// TwinCAT 3 PLC project Untitled1
// ProgramVersion: 3.1.4024.0
// libraries:
//   Tc2_Standard, * (Beckhoff Automation GmbH)
//   Tc2_System, * (Beckhoff Automation GmbH)
//   Tc3_Module, * (Beckhoff Automation GmbH)
// project tree:
//   GVLs/ GVL_IO.TcGVL
//   / PlcTask.TcTTO
//   POUs/ MAIN.TcPOU
// real-time tasks:
//   TASK PlcTask: cycle T#10ms, priority 20, ADS port 350
// I/O:
//   DEVICE Device 2 (EtherCAT), AmsNetId 169.254.197.213.3.1
//     Term 1 (EK1100) [EK1100 EtherCAT Coupler (2A E-Bus)]
//       Term 2 (EL1008) [EL1008 8Ch. Dig. Input 24V, 3ms]
//       Term 3 (EL3064) [EL3064 4Ch. Ana. Input 0-10V]
//       Term 4 (EL4034) [EL4034 4Ch. Ana. Output +/-10V, 12bit]
//       Term 5 (EL9011) [EL9011 End Terminal]
// variable links:
//   Untitled1/Untitled1 Instance <-> Device 2 (EtherCAT)/Term 1 (EK1100)/Term 2 (EL1008)
//     PlcTask Inputs/GVL_IO.bDoorInerlock <-> Channel 5/GVL_IO.bDoorInerlock
//     PlcTask Inputs/GVL_IO.bLeftPinLockSens <-> Channel 3/GVL_IO.bLeftPinLockSens
//     PlcTask Inputs/GVL_IO.bLeftPistonSens <-> Channel 2/GVL_IO.bLeftPistonSens
//     PlcTask Inputs/GVL_IO.bRightPinLockSens <-> Channel 4/GVL_IO.bRightPinLockSens
//     PlcTask Inputs/GVL_IO.nRightPistonSens <-> Channel 1/GVL_IO.nRightPistonSens
//   Untitled1/Untitled1 Instance <-> Device 2 (EtherCAT)/Term 1 (EK1100)/Term 3 (EL3064)
//     PlcTask Inputs/GVL_IO.rCurrentHW <-> AI Standard Channel 1/GVL_IO.rCurrentHW
//   Untitled1/Untitled1 Instance <-> Device 2 (EtherCAT)/Term 1 (EK1100)/Term 4 (EL4034)
//     PlcTask Outputs/GVL_IO.iMotorPowerHW <-> AO Outputs Channel 2/GVL_IO.iMotorPowerHW
//     PlcTask Outputs/GVL_IO.iSetPistonsPressureHW <-> AO Outputs Channel 1/GVL_IO.iSetPistonsPressureHW

CONFIGURATION Untitled1
    RESOURCE PLC ON TwinCAT3
        TASK PlcTask(INTERVAL := T#10ms, PRIORITY := 20);
        PROGRAM MAIN WITH PlcTask : MAIN;
    END_RESOURCE
END_CONFIGURATION

// ---- GVLs/GVL_IO.TcGVL

VAR_GLOBAL
	rCurrentHW				AT%I*	:	INT;
	iPistonsPressureHW		AT%I* 	:	INT;
	bRightPinLockSens		AT%I*	:	BOOL;
	bLeftPinLockSens		AT%I*	:	BOOL;
	bLeftPistonSens			AT%I*	: 	BOOL;
	nRightPistonSens		AT%I*	:	BOOL;
	bDoorInerlock			AT%I*	:	BOOL;
	
	iSetPistonsPressureHW	AT%Q* 	:	INT;
	iMotorPowerHW			AT%Q*	:	INT;
	iLeftPinForce			AT%I* 	:	INT;
	iRightPinForce			AT%I* 	:	INT;
	
END_VAR

// ---- POUs/MAIN.TcPOU
PROGRAM MAIN
VAR
	ProcessTime			:	TON;
	RunTimer			:	TON;
	StopTimer			:	TON;
	HoldTimer			:	TON;
	
	iHighPower			: 	INT;
	iHoldPower			: 	INT;
	TestState			:	INT;
	CSVstate			:	INT;
	iMotorPower			:	INT;
	iTestCounter		:	INT;
	iCycleToRun			:	UDINT;
	iPistonsPressure	:	INT;
	
	bStartTest			:	BOOL;
	bStopTest			:	BOOL;
	bTimeoutError		: 	BOOL;
	bProcessEndAtPins	: 	BOOL;
	bProcessEndAtTimeout: 	BOOL;
	bAutomatedOperation	:	BOOL;
	bWriteDataEnd		: 	BOOL;
	bReadyToRun			: 	BOOL;
	
	rMotorCurrenr		:	REAL;
	rRecordMotorCurrenr	:	REAL; //csv
	rTimeToStop			: 	REAL;
	rHMI_MotorCurrent	: 	REAL;// By mA
	rRightPinForce		:	REAL;
	rLeftPinForce		:	REAL;
	iPistonsForceHMI	:	INT;
	
	
	
	arrCurrentMessure	:	ARRAY[1..100] OF REAL;
	arrLeftPinMessure	:	ARRAY[1..100] OF REAL;
	arrRightPinMessure	:	ARRAY[1..100] OF REAL;
	i					:	INT;

	sDataToWrite		:	STRING[500];
	fbFileOpen      	: 	FB_FileOpen;
	fbFileWrite      	:	FB_FileWrite;
	fbFileClose       	: 	FB_FileClose;
	bKeepRuningTests: BOOL;
END_VAR

IF bDoorInerlock THEN
	RunTest();
	SaveData();
END_IF

iSetPistonsPressureHW:=REAL_TO_INT(INT_TO_REAL(iPistonsForceHMI)*32.59);
rMotorCurrenr:=(INT_TO_REAL(rCurrentHW)/32767.0)*15.0;
rHMI_MotorCurrent:=rMotorCurrenr*1000;
iMotorPowerHW:=real_to_int((INT_TO_REAL(iMotorPower)/100)*16383);

ACTION RunTest:
ProcessTime(IN:= , PT:=T#2500MS , Q=> , ET=> );
RunTimer(IN:= , PT:=T#450MS , Q=> , ET=> );
StopTimer(IN:= , PT:=T#50MS , Q=> , ET=> );
HoldTimer(IN:= , PT:=T#2S , Q=> , ET=> );
IF TestState=0 AND CSVstate=0 THEN
	bReadyToRun:=TRUE;
ELSE 
	bReadyToRun:=FALSE;
END_IF
IF iTestCounter<=iCycleToRun THEN
	bKeepRuningTests:=TRUE;
ELSE
	bKeepRuningTests:=FALSE;	
END_IF



CASE TestState OF
	0://standby
		ProcessTime.IN:=FALSE;
		IF bStartTest AND NOT bStopTest AND bLeftPistonSens AND nRightPistonSens THEN
			IF NOT bAutomatedOperation THEN
				bStartTest:=FALSE;
			END_IF
			iTestCounter:=iTestCounter+1;
			ProcessTime.IN:=TRUE;
			bProcessEndAtPins:=FALSE;
			bProcessEndAtTimeout:=FALSE;
			//bReadyToRun:=FALSE;
			i:=1;
			TestState:=10;
		END_IF
	
	10:// start movment and reach pins lock sensors
		arrCurrentMessure[i]:=rMotorCurrenr;
		arrLeftPinMessure[i]:=iLeftPinForce;
		arrRightPinMessure[i]:=iRightPinForce;
		i:=i+1;
		IF i>100 THEN
			i:=1;
		END_IF
		RunTimer.IN:=TRUE;
		iMotorPower:=iHighPower;
		
		IF bLeftPinLockSens AND bRightPinLockSens THEN
			bProcessEndAtPins:=TRUE;
			RunTimer.IN:=FALSE;
			iMotorPower:=iHoldPower;	
			//StopTimer.IN:=TRUE;			
			TestState:=20;
		ELSIF RunTimer.Q THEN
			bProcessEndAtTimeout:=TRUE;
			RunTimer.IN:=FALSE;
			iMotorPower:=0;				
			TestState:=40;
		END_IF	
		
	20: //hols pins in open position for 2 sec
		HoldTimer.IN:=TRUE;
		IF HoldTimer.Q THEN
			iMotorPower:=0;
			TestState:=30;
			FOR i:=i TO i-5 DO
				rRecordMotorCurrenr:=(rRecordMotorCurrenr+arrCurrentMessure[i])/5;
				rRightPinForce:=(rRightPinForce+arrLeftPinMessure[i])/5;	
				rLeftPinForce:=(rLeftPinForce+arrRightPinMessure[i])/5;	
			END_FOR			
		END_IF

		
	
	30:// end movment, release motor until pins in close position
		IF bLeftPistonSens AND nRightPistonSens THEN
			rTimeToStop:=TIME_TO_REAL(StopTimer.ET);
			TestState:=40;
		END_IF

	40:// write data to csv
		IF bWriteDataEnd THEN
			TestState:=0;
		END_IF
END_CASE

IF ProcessTime.Q THEN
	bTimeoutError:=TRUE;
ELSE
	bTimeoutError:=FALSE;	
END_IF
END_ACTION

ACTION SaveData:
sDataToWrite:=concat(REAL_TO_STRING(rRightPinForce),concat(',',concat(REAL_TO_STRING(rLeftPinForce),concat(',',concat(REAL_TO_STRING(rRecordMotorCurrenr),concat(',',concat(REAL_TO_STRING(rTimeToStop),concat(',',concat(BOOL_TO_STRING(bProcessEndAtPins),concat(',',concat(INT_TO_STRING(iPistonsForceHMI),'$N')))))))))));
fbFileOpen(
	sNetId:='' , 
	sPathName:='C:\Users\Administrator\Desktop\Logs\Tests.csv ', // add controller path
	nMode:=FOPEN_MODEAPPEND , 
	ePath:= , 
	bExecute:= , 
	tTimeout:=T#3S , 
	bBusy=> , 
	bError=> , 
	nErrId=> , 
	hFile=> );
fbFileWrite(
	sNetId:='' , 
	hFile:=fbFileOpen.hFile , 
	pWriteBuff:=ADR(sDataToWrite) , 
	cbWriteLen:=LEN(sDataToWrite) , 
	bExecute:= , 
	tTimeout:=T#3S , 
	bBusy=> , 
	bError=> , 
	nErrId=> , 
	cbWrite=> );
fbFileClose(
	sNetId:='' , 
	hFile:=fbFileOpen.hFile , 
	bExecute:= , 
	tTimeout:=T#3S , 
	bBusy=> , 
	bError=> , 
	nErrId=> );			

CASE CSVstate OF
	0://standby
	fbFileOpen.bExecute:=FALSE;
	fbFileWrite.bExecute:=FALSE;
	fbFileClose.bExecute:=FALSE;
		IF TestState=40 THEN
			CSVstate:=10;
		END_IF
	10:// open file
		fbFileOpen.bExecute:=TRUE;
		IF fbFileOpen.bBusy AND NOT fbFileOpen.bError THEN
			CSVstate:=15;
		END_IF	
	15:		
		IF NOT fbFileOpen.bError AND NOT fbFileOpen.bBusy THEN
			CSVstate:=20;
		END_IF	
	20:// write data
		fbFileWrite.bExecute:=TRUE;
		IF fbFileWrite.bBusy AND NOT fbFileWrite.bError THEN
			CSVstate:=25;
		END_IF		
	25:
		IF NOT fbFileWrite.bError AND NOT fbFileWrite.bBusy THEN
			CSVstate:=30;
		END_IF	
	30:// close file
		fbFileClose.bExecute:=TRUE;
		IF fbFileClose.bBusy AND NOT fbFileClose.bError THEN
			CSVstate:=35;
		END_IF			
	35:
		IF NOT fbFileClose.bError AND NOT fbFileClose.bBusy THEN
			CSVstate:=0;
			bWriteDataEnd:=TRUE;
		END_IF
	
END_CASE
END_ACTION

ACTION SideTest:

RunTimer(IN:= , PT:=T#1S , Q=> , ET=> );
StopTimer(IN:= , PT:=T#500MS , Q=> , ET=> );

CASE TestState OF
	0://standby
	StopTimer.IN:=FALSE;	
	RunTimer.IN:=FALSE;
		IF bStartTest THEN
			TestState:=10;
		END_IF
	
	10:// start movment

		RunTimer.IN:=TRUE;
		iMotorPower:=30;
		
		IF RunTimer.Q THEN
			RunTimer.IN:=FALSE;
			iMotorPower:=0;	
			TestState:=20;
		END_IF	
	
	20:// end movment
		StopTimer.IN:=TRUE;	
		IF 	StopTimer.Q THEN
			TestState:=0;
		END_IF


END_CASE
END_ACTION

END_PROGRAM
